TYPE st_Enclosure_params :
STRUCT
	climate			: ST_EnclosureClimate_params;
	ledstrip		: st_Ledstrip_params;
END_STRUCT
END_TYPE

(* stored: Version 1.1.0.1, ProductVersion 3.1.4026.18
   DUT st_Enclosure_params: Id {1e450fc7-8564-4e20-a076-940e16d24ad4} *)
